// TIA Portal project "MyAwesomeTIAproject_v5" (V19)

(* hardware
DEVICE "PLC_1"  S7-1200 Station
   slot 0: "Rack_0"  S7-1200 Rack  Rack  V1.0
   slot 1: "PLC_1"  CPU 1212C DC/DC/DC  6ES7 212-1AE40-0XB0  V4.6
*)

// ===== PLC "PLC_1"  CPU 1212C DC/DC/DC =====

TYPE "Crossroad_Input"
   STRUCT
      btnStart : Bool := FALSE;
      btnPause : Bool := FALSE;
      btnStop : Bool := FALSE;
      btnCrosswalk1 : Bool := FALSE;
      btnCrosswalk2 : Bool := FALSE;
   END_STRUCT;
END_TYPE

TYPE "Crossroad_Output"
   STRUCT
      crossroadType : Bool := FALSE;
      trafficLightGreen1 : Bool := FALSE;
      trafficLightsYellow1 : Bool := FALSE;
      trafficLightsRed1 : Bool := FALSE;
      trafficLightGreen2 : Bool := FALSE;
      trafficLightsYellow2 : Bool := FALSE;
      trafficLightsRed2 : Bool := FALSE;
      pedestrianLightGreen1 : Bool := FALSE;
      pedestrianLightRed1 : Bool := FALSE;
      pedestrianLightGreen2 : Bool := FALSE;
      pedestrianLightRed2 : Bool := FALSE;
   END_STRUCT;
END_TYPE

DATA_BLOCK "DB_ProcessData"   // DB1
{ S7_Optimized_Access := 'TRUE' }
VERSION : 0.1
   VAR
      input : "Crossroad_Input";
      output : "Crossroad_Output";
   END_VAR
BEGIN
END_DATA_BLOCK

ORGANIZATION_BLOCK "Main"   // OB1, LAD, ProgramCycle
TITLE = "Main Program Sweep (Cycle)"
{ S7_Optimized_Access := 'TRUE' }
VERSION : 0.1
   VAR_INPUT
      Initial_Call : Bool;   // Initial call of this OB
      Remanence : Bool;   // =True, if remanent data are available
   END_VAR
BEGIN
END_ORGANIZATION_BLOCK